{attribute addProperty BoxType "KL3224"}
{attribute addProperty Id "Channel_1Channel_B0A8062F00Channel_2Channel_B0A8062F00Channel_3Channel_B0A8062F00Channel_4Channel_B0A8062F00"}
{attribute addProperty CRC "2945616803"}
{attribute addProperty SizeInBites "0"}
{attribute addProperty SizeInBytes "0"}
TYPE KL3224_AF928BA3 :
STRUCT
	{attribute addProperty Name "Channel_1"}
	Channel_1 : Channel_B0A8062F;
	{attribute addProperty Name "Channel_2"}
	Channel_2 : Channel_B0A8062F;
	{attribute addProperty Name "Channel_3"}
	Channel_3 : Channel_B0A8062F;
	{attribute addProperty Name "Channel_4"}
	Channel_4 : Channel_B0A8062F;
END_STRUCT
END_TYPE

(* stored: Version 1.2.0.0, ProductVersion 3.1.4024.9
   DUT KL3224_AF928BA3: Id {366afac6-77ed-4090-99ed-d8b394dbd8ae} *)
